TYPE ST_Data :
STRUCT
	rSystemOutVoltageDc		: REAL;		// CMD 01
	rSystemOutCurrentDc		: REAL;		// CMD 01
	rNumberOfModules		: REAL;		// CMD 02
	stModuleData			: ARRAY [0..10] OF ST_ModuleData;
	
	
	
	
	
END_STRUCT
END_TYPE

(* stored: Version 1.1.0.1, ProductVersion 3.1.4026.18
   DUT ST_Data: Id {02434dd0-cfd4-4924-af25-fcf438e2dcda} *)
